FUNCTION_BLOCK T_BaseMode IMPLEMENTS I_PackMode
VAR_INPUT
END_VAR
VAR_OUTPUT
END_VAR
VAR
END_VAR

{warning 'add method implementation '}
METHOD Aborted
END_METHOD

{warning 'add method implementation '}
METHOD Aborting
END_METHOD

{warning 'add method implementation '}
METHOD Clearing
END_METHOD

{warning 'add method implementation '}
METHOD Complete
END_METHOD

{warning 'add method implementation '}
METHOD Completing
END_METHOD

{warning 'add method implementation '}
METHOD Execute
END_METHOD

{warning 'add method implementation '}
METHOD Held
END_METHOD

{warning 'add method implementation '}
METHOD Holding
END_METHOD

{warning 'add method implementation '}
METHOD Idle
END_METHOD

{warning 'add method implementation '}
METHOD Resetting
END_METHOD

{warning 'add method implementation '}
METHOD Starting
END_METHOD

{warning 'add method implementation '}
METHOD Stopped
END_METHOD

{warning 'add method implementation '}
METHOD Stopping
END_METHOD

{warning 'add method implementation '}
METHOD Suspended
END_METHOD

{warning 'add method implementation '}
METHOD Suspending
END_METHOD

{warning 'add method implementation '}
METHOD Unholding
END_METHOD

{warning 'add method implementation '}
METHOD Unsuspending
END_METHOD

END_FUNCTION_BLOCK

(* stored: Version 1.1.0.1, ProductVersion 3.1.4024.12
   POU T_BaseMode: Id {e529a071-6118-4f9e-bb57-081bd478720f}, SpecialFunc None
   Folder ActingStates: Id {07ad3554-1045-41d8-8cba-5fe80924805e}
   Folder Properties: Id {c547770d-106f-4617-b0d0-830f34c2f4dd}
   Folder WaitingStates: Id {091b64c0-263b-4a2f-8509-64b92535fb4b}
   Method Aborted: Id {ff791c37-6c7c-4fdc-8617-29f763dc48d7}
   Method Aborting: Id {3e8e7892-4bb0-4922-8a9a-015c48efff1e}
   Method Clearing: Id {f4ac0fe3-c9c8-4544-88d2-f7b6c093c564}
   Method Complete: Id {3a077633-d3ce-441a-b7ad-0f2144b1d9fb}
   Method Completing: Id {c2540e52-6719-4b0c-9487-f6d5ca2f6df0}
   Method Execute: Id {201854c4-3d73-4adf-a610-f5dc16a9cee0}
   Method Held: Id {9b80ca93-f07a-45e0-8d8a-40221f4762bb}
   Method Holding: Id {f59b21da-86ac-4af6-84a8-c8dd65f726c9}
   Method Idle: Id {f7af9414-0967-4ea0-b37d-1eeb0473981f}
   Method Resetting: Id {609fa116-bf8e-4353-a766-58f5a27b7db1}
   Method Starting: Id {5541f051-747b-4c88-b64b-e8084a973b8d}
   Method Stopped: Id {6c9ec9e7-0db5-4794-ab34-0a245c70829a}
   Method Stopping: Id {04a30b4b-4964-4f78-ba85-120e4cc19813}
   Method Suspended: Id {99866019-09d0-4ca3-a85c-1f9199160951}
   Method Suspending: Id {55e031be-a07e-4434-b673-0d84f4347e3a}
   Method Unholding: Id {b01b9486-4a69-49ed-a4fc-6be449ee33fa}
   Method Unsuspending: Id {ed108570-a1e9-4f83-9df2-6b8b4e25505a} *)
